(* Logix 5000 project; controller PRU vendor 1 type 14 code 107 rev 20.13; software revision 20.01; part 11 of 17 *)
(* tags used below, declared in another part *)
   AFI : BOOL;
   CHANGING_TOTE : BOOL;
   CHANGING_TOTE_1 : BOOL;
   CHANGING_TOTE_2 : BOOL;
   CHANGING_TOTE_3 : BOOL;
   CHANGING_TOTE_4 : BOOL;
   CHANGING_TOTE_5 : BOOL;
   COOL_VFD_Message : MESSAGE;
   DI0_ION : BOOL;
   DI10_ION : BOOL;
   DI11_ION : BOOL;
   DI12_ION : BOOL;
   DI13_ION : BOOL;
   DI14_ION : BOOL;
   DI15_ION : BOOL;
   DI16_ION : BOOL;
   DI17_ION : BOOL;
   DI18_ION : BOOL;
   DI19_ION : BOOL;
   DI1_ION : BOOL;
   DI20_ION : BOOL;
   DI21_ION : BOOL;
   DI22_ION : BOOL;
   DI23_ION : BOOL;
   DI24_ION : BOOL;
   DI25_ION : BOOL;
   DI26_ION : BOOL;
   DI27_ION : BOOL;
   DI28_ION : BOOL;
   DI29_ION : BOOL;
   DI2_ION : BOOL;
   DI30_ION : BOOL;
   DI31_ION : BOOL;
   DI3_ION : BOOL;
   DI4_ION : BOOL;
   DI5_ION : BOOL;
   DI6_ION : BOOL;
   DI7_ION : BOOL;
   DI8_ION : BOOL;
   DI9_ION : BOOL;
   DUMMY_REAL : REAL;
   ESR_CONTACT_1_ION : BOOL;
   ESR_CONTACT_2_ION : BOOL;
   ESR_CONTACT_3_ION : BOOL;
   ESR_RESET_PB_ION : BOOL;
   ESTOP_PB_IOF : BOOL;   // E-STOP PUSHBUTTON IS PUSHED.
   FAULT : DINT[100];
   FS0101_ION : BOOL;   // LOW FLOW SWITCH - INLET AND DISCHARGE PURGE
   FS0102H_ION : BOOL;   // HIGH FLOW SWITCH - DISCHARGE END SHAFT SEAL
   FS0102L_ION : BOOL;   // LOW FLOW SWITCH - DISCHARGE END SHAFT SEAL
   FS0103H_ION : BOOL;   // HIGH FLOW SWITCH - CHAMBER END INLET SEALS
   FS0103L_ION : BOOL;   // LOW FLOW SWITCH - CHAMBER END INLET SEALS
   FS0201_ION : BOOL;   // LOW FLOW SWITCH - KG021 PURGE
   FS0202_ION : BOOL;   // LOW FLOW SWITCH - KG022 PURGE
   FS0203H_ION : BOOL;   // HIGH FLOW SWITCH - COOLING SHAFT SEALS
   FS0203L_ION : BOOL;   // LOW FLOW SWITCH - COOLING SHAFT SEALS
   FS0204_ION : BOOL;   // LOW FLOW SWITCH - COOLING SCREW COOLING WATER
   HEATER_1_ALARM_ION : BOOL;
   HEATER_2_ALARM_ION : BOOL;
   HEATER_3_ALARM_ION : BOOL;
   HEATER_4_ALARM_ION : BOOL;
   HEATER_5_ALARM_ION : BOOL;
   HMI_ALARM_RESET : BOOL;
   HMI_ALARM_RESET_ONS : BOOL;
   HMI_ALARM_RESET_PB : BOOL;
   HMI_ALARM_RESET_TOF : TIMER;
   HMI_ALARM_RESET_TON : TIMER;
   HMI_COOL_MOTOR : INT;
   HMI_COOL_MOTOR_PRE : INT;
   HMI_DI0_FORCE_OFF : BOOL;
   HMI_DI0_FORCE_ON : BOOL;
   HMI_DI10_FORCE_OFF : BOOL;
   HMI_DI10_FORCE_ON : BOOL;
   HMI_DI11_FORCE_OFF : BOOL;
   HMI_DI11_FORCE_ON : BOOL;
   HMI_DI12_FORCE_OFF : BOOL;
   HMI_DI12_FORCE_ON : BOOL;
   HMI_DI13_FORCE_OFF : BOOL;
   HMI_DI13_FORCE_ON : BOOL;
   HMI_DI14_FORCE_OFF : BOOL;
   HMI_DI14_FORCE_ON : BOOL;
   HMI_DI15_FORCE_OFF : BOOL;
   HMI_DI15_FORCE_ON : BOOL;
   HMI_DI16_FORCE_OFF : BOOL;
   HMI_DI16_FORCE_ON : BOOL;
   HMI_DI17_FORCE_OFF : BOOL;
   HMI_DI17_FORCE_ON : BOOL;
   HMI_DI18_FORCE_OFF : BOOL;
   HMI_DI18_FORCE_ON : BOOL;
   HMI_DI19_FORCE_OFF : BOOL;
   HMI_DI19_FORCE_ON : BOOL;
   HMI_DI1_FORCE_OFF : BOOL;
   HMI_DI1_FORCE_ON : BOOL;
   HMI_DI20_FORCE_OFF : BOOL;
   HMI_DI20_FORCE_ON : BOOL;
   HMI_DI21_FORCE_OFF : BOOL;
   HMI_DI21_FORCE_ON : BOOL;
   HMI_DI22_FORCE_OFF : BOOL;
   HMI_DI22_FORCE_ON : BOOL;
   HMI_DI23_FORCE_OFF : BOOL;
   HMI_DI23_FORCE_ON : BOOL;
   HMI_DI24_FORCE_OFF : BOOL;
   HMI_DI24_FORCE_ON : BOOL;
   HMI_DI25_FORCE_OFF : BOOL;
   HMI_DI25_FORCE_ON : BOOL;
   HMI_DI26_FORCE_OFF : BOOL;
   HMI_DI26_FORCE_ON : BOOL;
   HMI_DI27_FORCE_OFF : BOOL;
   HMI_DI27_FORCE_ON : BOOL;
   HMI_DI28_FORCE_OFF : BOOL;
   HMI_DI28_FORCE_ON : BOOL;
   HMI_DI29_FORCE_OFF : BOOL;
   HMI_DI29_FORCE_ON : BOOL;
   HMI_DI2_FORCE_OFF : BOOL;
   HMI_DI2_FORCE_ON : BOOL;
   HMI_DI30_FORCE_OFF : BOOL;
   HMI_DI30_FORCE_ON : BOOL;
   HMI_DI31_FORCE_OFF : BOOL;
   HMI_DI31_FORCE_ON : BOOL;
   HMI_DI3_FORCE_OFF : BOOL;
   HMI_DI3_FORCE_ON : BOOL;
   HMI_DI4_FORCE_OFF : BOOL;
   HMI_DI4_FORCE_ON : BOOL;
   HMI_DI5_FORCE_OFF : BOOL;
   HMI_DI5_FORCE_ON : BOOL;
   HMI_DI6_FORCE_OFF : BOOL;
   HMI_DI6_FORCE_ON : BOOL;
   HMI_DI7_FORCE_OFF : BOOL;
   HMI_DI7_FORCE_ON : BOOL;
   HMI_DI8_FORCE_OFF : BOOL;
   HMI_DI8_FORCE_ON : BOOL;
   HMI_DI9_FORCE_OFF : BOOL;
   HMI_DI9_FORCE_ON : BOOL;
   HMI_DML_MOTOR : INT;
   HMI_DML_MOTOR_PRE : INT;
   HMI_DMR_MOTOR : INT;
   HMI_DMR_MOTOR_PRE : INT;
   K0621_ALARM_ION : BOOL;
   K0621_IS_CLOSED : BOOL;
   K0621_IS_LOCAL : BOOL;
   K0621_IS_OPEN : BOOL;
   K0621_IS_REMOTE : BOOL;
   K0622_ALARM_ION : BOOL;
   K0622_IS_CLOSED : BOOL;
   K0622_IS_LOCAL : BOOL;
   K0622_IS_OPEN : BOOL;
   K0622_IS_REMOTE : BOOL;
   MSG_ONS3 : BOOL;
   ONE_SEC : BOOL;   // 50% Duty Cycle
   ONE_SEC_ONS : BOOL;
   ONE_SEC_SS : BOOL;
   PLC_Time : DINT[8];
   PS0101_ION : BOOL;   // PRESSURE SWITCH - CONTROL PANEL Y/Z N2 PURGE
   PS0102_ION : BOOL;   // PRESSURE SWITCH - MAIN N2 SUPPLY
   PVTIME_OSC_1 : TIMER;
   PVTIME_OSC_2 : TIMER;
   PVTIME_UPDATE : BOOL;
   RESUME_DISCHARGE : BOOL;
   START_TOTE_CHANGE : BOOL;
   TE0101 : REAL;
   TE0101_SEL_ION : BOOL;
   TE0102 : REAL;
   TE0102_SEL_ION : BOOL;
   TE0103 : REAL;
   TE0103_SEL_ION : BOOL;
   TE0104 : REAL;
   TE0104_SEL_ION : BOOL;
   TE0105 : REAL;
   TE0105_SEL_ION : BOOL;
   TE0106 : REAL;
   TE0106_SEL_ION : BOOL;
   TE0107 : REAL;
   TE0107_SEL_ION : BOOL;
   TE0108 : REAL;
   TE0108_SEL_ION : BOOL;
   TE0109 : REAL;
   TE0109_SEL_ION : BOOL;
   TE0110 : REAL;
   TE0110_SEL_ION : BOOL;
   TE0111 : REAL;
   TE0111_SEL_ION : BOOL;
   TE0112 : REAL;
   TE0112_SEL_ION : BOOL;
   TE0113 : REAL;
   TE0113_SEL_ION : BOOL;
   TE0114 : REAL;
   TE0114_SEL_ION : BOOL;
   TE0115 : REAL;
   TE0115_SEL_ION : BOOL;
   TE0116 : REAL;
   TE0116_SEL_ION : BOOL;
   TE0117 : REAL;
   TE0117_SEL_ION : BOOL;
   TE0118 : REAL;
   TE0118_SEL_ION : BOOL;
   TE0119 : REAL;
   TE0119_SEL_ION : BOOL;
   TE0120 : REAL;
   TE0120_SEL_ION : BOOL;
   TE0121 : REAL;
   TE0121_SEL_ION : BOOL;
   TE0122 : REAL;
   TE0122_SEL_ION : BOOL;
   TE0123 : REAL;
   TE0123_SEL_ION : BOOL;
   TE0124 : REAL;
   TE0124_SEL_ION : BOOL;
   TE0125 : REAL;
   TE0125_SEL_ION : BOOL;
   TE0126 : REAL;
   TE0126_SEL_ION : BOOL;
   TE0127 : REAL;
   TE0127_SEL_ION : BOOL;
   TE0128 : REAL;
   TE0128_SEL_ION : BOOL;
   TE0129 : REAL;
   TE0129_SEL_ION : BOOL;
   TE0130 : REAL;
   TE0130_SEL_ION : BOOL;
   TIMER_MSG_OFF : TIMER;
   TIMER_MSG_ON : TIMER;
   TIMER_ONE_SEC_OFF : TIMER;
   TIMER_ONE_SEC_ON : TIMER;
   TIMER_WDT_OFF : TIMER;
   TIMER_WDT_ON : TIMER;
   TOTE_CHANGE_MODE : INT;
   TOTE_CHANGE_REMAINING : REAL;
   TOTE_CHANGE_TIMED_OUT : BOOL;
   TOTE_CHANGEOUT_TOF : TIMER;
   TOTE_CHANGEOUT_TON : TIMER;
   VFD_3_Current : DINT;
   VFD_3_Current_Real : REAL;
   VFD_3_Tot : EnergyTot;   // Cooling Screw
   VFD_AUTO_RESET : BOOL;
   WDT_ONS : BOOL;
   WDT_SS : BOOL;
   ZONE_1_SELECT_TE : TE_SELECTED_AVE;
   ZONE_1_TEMP_AVE : DINT;
   ZONE_2_SELECT_TE : TE_SELECTED_AVE;
   ZONE_2_TEMP_AVE : REAL;
   ZONE_3_SELECT_TE : TE_SELECTED_AVE;
   ZONE_3_TEMP_AVE : REAL;
   ZONE_4_SELECT_TE : TE_SELECTED_AVE;
   ZONE_4_TEMP_AVE : REAL;
   ZONE_5_SELECT_TE : TE_SELECTED_AVE;
   ZONE_5_TEMP_AVE : REAL;
   ZONE_6_SELECT_TE : TE_SELECTED_AVE;
   ZONE_6_TEMP_AVE : REAL;
   ZONE_7_SELECT_TE : TE_SELECTED_AVE;
   ZONE_7_TEMP_AVE : REAL;
(* MainProgram, continued *)

ROUTINE C04_ZONE_TEMPS   (* ladder *)
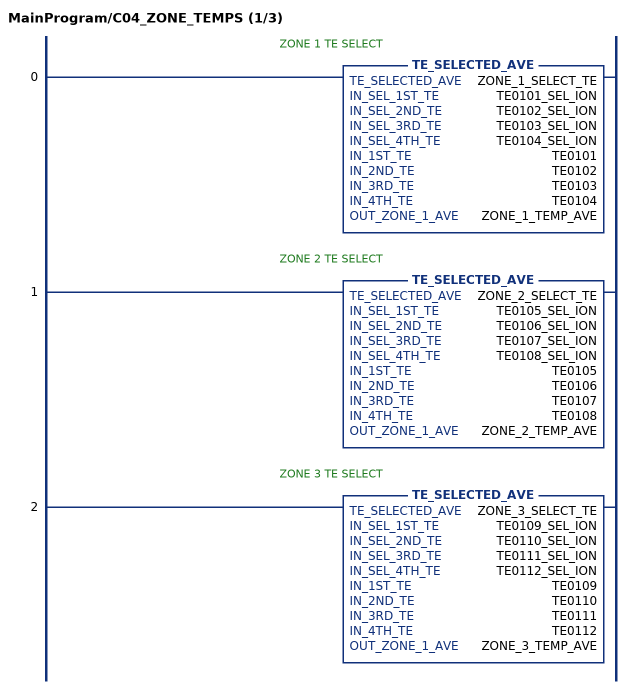
   // ZONE 1 TE SELECT
   0: TE_SELECTED_AVE(ZONE_1_SELECT_TE,TE0101_SEL_ION,TE0102_SEL_ION,TE0103_SEL_ION,TE0104_SEL_ION,TE0101,TE0102,TE0103,TE0104,ZONE_1_TEMP_AVE);
   // ZONE 2 TE SELECT
   1: TE_SELECTED_AVE(ZONE_2_SELECT_TE,TE0105_SEL_ION,TE0106_SEL_ION,TE0107_SEL_ION,TE0108_SEL_ION,TE0105,TE0106,TE0107,TE0108,ZONE_2_TEMP_AVE);
   // ZONE 3 TE SELECT
   2: TE_SELECTED_AVE(ZONE_3_SELECT_TE,TE0109_SEL_ION,TE0110_SEL_ION,TE0111_SEL_ION,TE0112_SEL_ION,TE0109,TE0110,TE0111,TE0112,ZONE_3_TEMP_AVE);
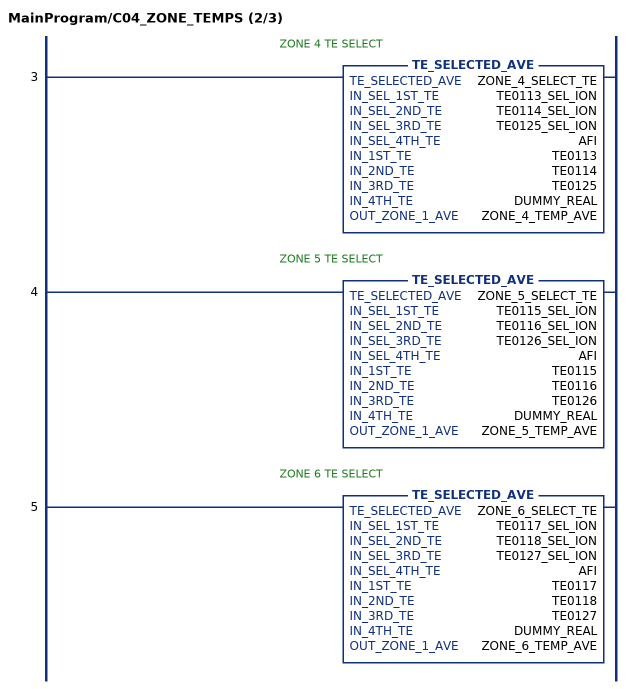
   // ZONE 4 TE SELECT
   3: TE_SELECTED_AVE(ZONE_4_SELECT_TE,TE0113_SEL_ION,TE0114_SEL_ION,TE0125_SEL_ION,AFI,TE0113,TE0114,TE0125,DUMMY_REAL,ZONE_4_TEMP_AVE);
   // ZONE 5 TE SELECT
   4: TE_SELECTED_AVE(ZONE_5_SELECT_TE,TE0115_SEL_ION,TE0116_SEL_ION,TE0126_SEL_ION,AFI,TE0115,TE0116,TE0126,DUMMY_REAL,ZONE_5_TEMP_AVE);
   // ZONE 6 TE SELECT
   5: TE_SELECTED_AVE(ZONE_6_SELECT_TE,TE0117_SEL_ION,TE0118_SEL_ION,TE0127_SEL_ION,AFI,TE0117,TE0118,TE0127,DUMMY_REAL,ZONE_6_TEMP_AVE);
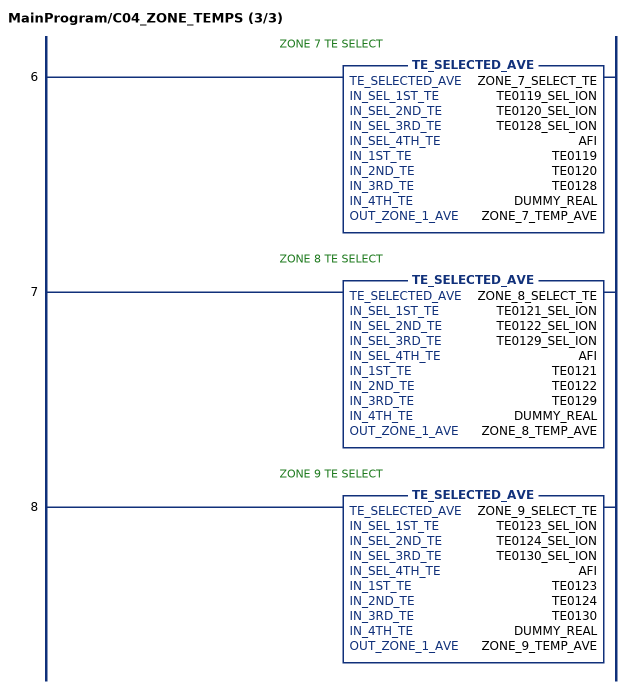
   // ZONE 7 TE SELECT
   6: TE_SELECTED_AVE(ZONE_7_SELECT_TE,TE0119_SEL_ION,TE0120_SEL_ION,TE0128_SEL_ION,AFI,TE0119,TE0120,TE0128,DUMMY_REAL,ZONE_7_TEMP_AVE);
   // ZONE 8 TE SELECT
   7: TE_SELECTED_AVE(ZONE_8_SELECT_TE,TE0121_SEL_ION,TE0122_SEL_ION,TE0129_SEL_ION,AFI,TE0121,TE0122,TE0129,DUMMY_REAL,ZONE_8_TEMP_AVE);
   // ZONE 9 TE SELECT
   8: TE_SELECTED_AVE(ZONE_9_SELECT_TE,TE0123_SEL_ION,TE0124_SEL_ION,TE0130_SEL_ION,AFI,TE0123,TE0124,TE0130,DUMMY_REAL,ZONE_9_TEMP_AVE);
END_ROUTINE

ROUTINE C05_TOTE_CHANGE   (* ladder *)
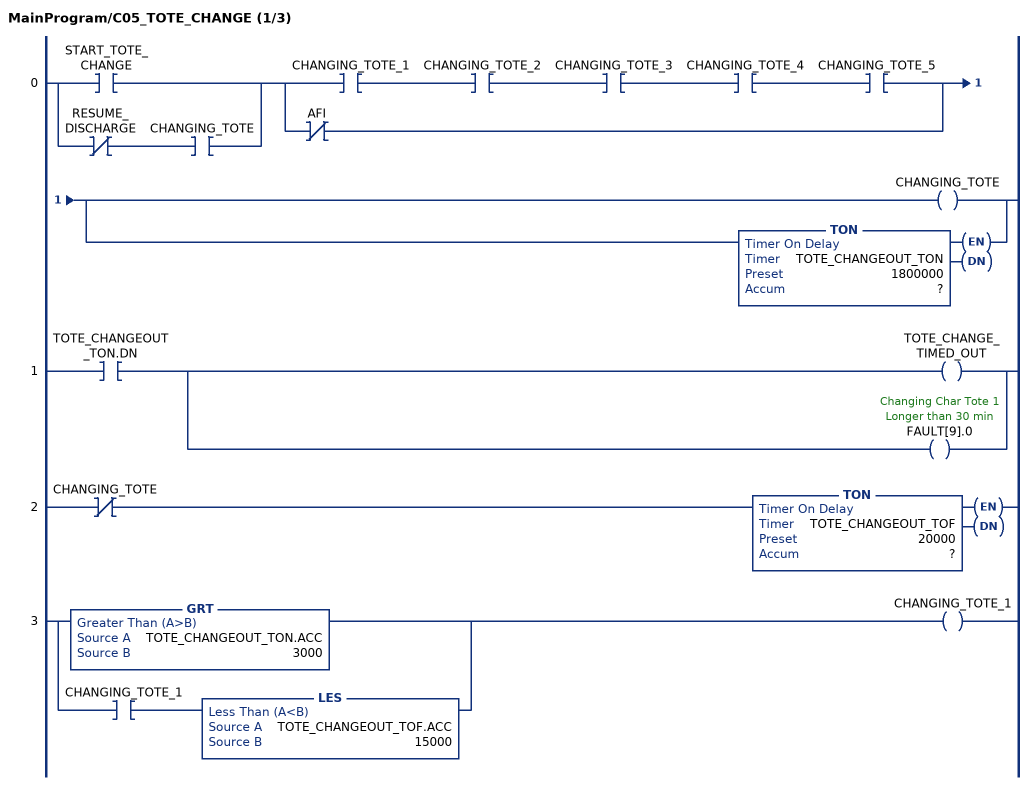
   0: [XIC(START_TOTE_CHANGE) ,XIO(RESUME_DISCHARGE) XIC(CHANGING_TOTE) ][XIC(CHANGING_TOTE_1) XIC(CHANGING_TOTE_2) XIC(CHANGING_TOTE_3) XIC(CHANGING_TOTE_4) XIC(CHANGING_TOTE_5) ,XIO(AFI) ][OTE(CHANGING_TOTE) ,TON(TOTE_CHANGEOUT_TON,?,?) ];
   1: XIC(TOTE_CHANGEOUT_TON.DN)[OTE(TOTE_CHANGE_TIMED_OUT) ,OTE(FAULT[9].0) ];
   2: XIO(CHANGING_TOTE)TON(TOTE_CHANGEOUT_TOF,?,?);
   3: [GRT(TOTE_CHANGEOUT_TON.ACC,3000) ,XIC(CHANGING_TOTE_1) LES(TOTE_CHANGEOUT_TOF.ACC,15000) ]OTE(CHANGING_TOTE_1);
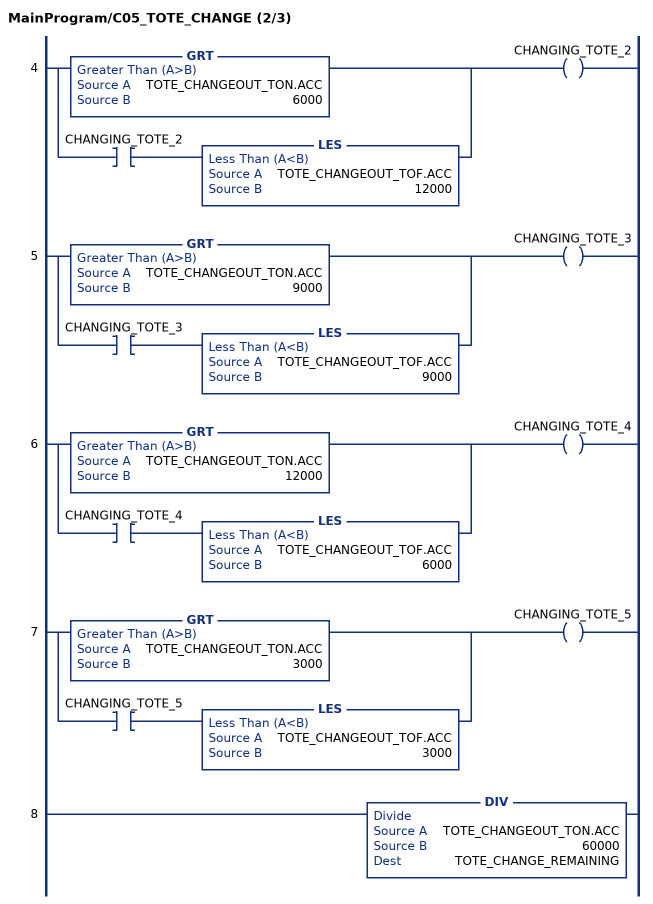
   4: [GRT(TOTE_CHANGEOUT_TON.ACC,6000) ,XIC(CHANGING_TOTE_2) LES(TOTE_CHANGEOUT_TOF.ACC,12000) ]OTE(CHANGING_TOTE_2);
   5: [GRT(TOTE_CHANGEOUT_TON.ACC,9000) ,XIC(CHANGING_TOTE_3) LES(TOTE_CHANGEOUT_TOF.ACC,9000) ]OTE(CHANGING_TOTE_3);
   6: [GRT(TOTE_CHANGEOUT_TON.ACC,12000) ,XIC(CHANGING_TOTE_4) LES(TOTE_CHANGEOUT_TOF.ACC,6000) ]OTE(CHANGING_TOTE_4);
   7: [GRT(TOTE_CHANGEOUT_TON.ACC,3000) ,XIC(CHANGING_TOTE_5) LES(TOTE_CHANGEOUT_TOF.ACC,3000) ]OTE(CHANGING_TOTE_5);
   8: DIV(TOTE_CHANGEOUT_TON.ACC,60000,TOTE_CHANGE_REMAINING);
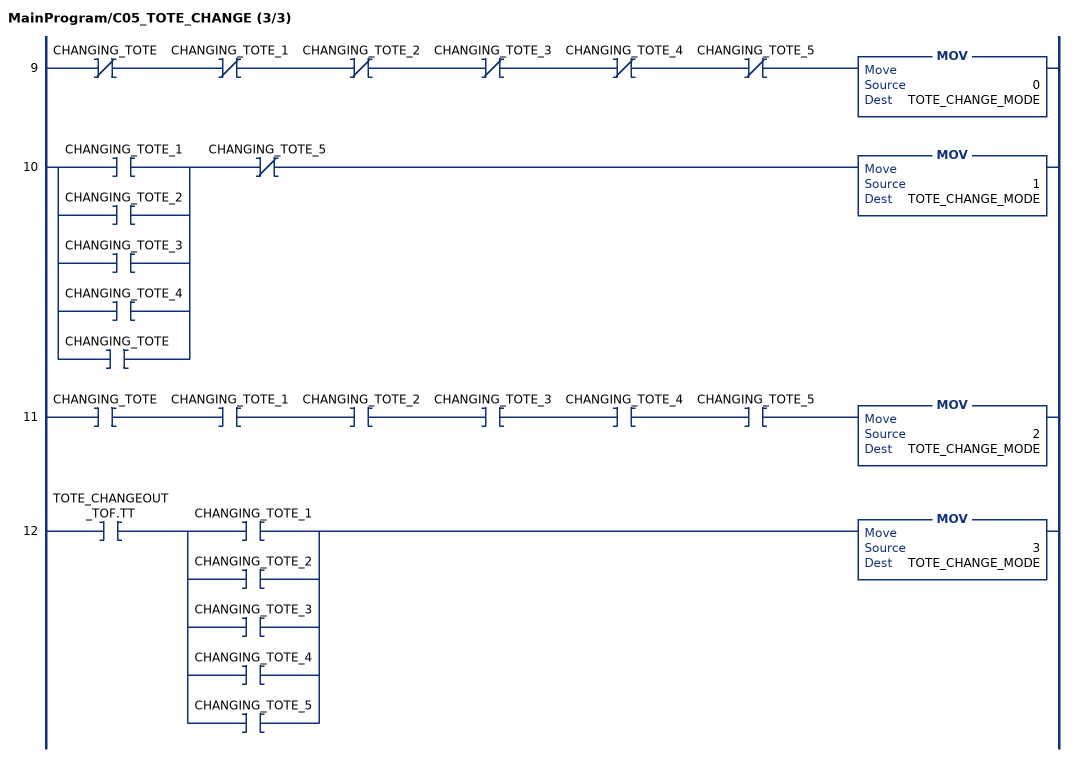
   9: XIO(CHANGING_TOTE)XIO(CHANGING_TOTE_1)XIO(CHANGING_TOTE_2)XIO(CHANGING_TOTE_3)XIO(CHANGING_TOTE_4)XIO(CHANGING_TOTE_5)MOV(0,TOTE_CHANGE_MODE);
   10: [XIC(CHANGING_TOTE_1) ,XIC(CHANGING_TOTE_2) ,XIC(CHANGING_TOTE_3) ,XIC(CHANGING_TOTE_4) ,XIC(CHANGING_TOTE) ]XIO(CHANGING_TOTE_5)MOV(1,TOTE_CHANGE_MODE);
   11: XIC(CHANGING_TOTE)XIC(CHANGING_TOTE_1)XIC(CHANGING_TOTE_2)XIC(CHANGING_TOTE_3)XIC(CHANGING_TOTE_4)XIC(CHANGING_TOTE_5)MOV(2,TOTE_CHANGE_MODE);
   12: XIC(TOTE_CHANGEOUT_TOF.TT)[XIC(CHANGING_TOTE_1) ,XIC(CHANGING_TOTE_2) ,XIC(CHANGING_TOTE_3) ,XIC(CHANGING_TOTE_4) ,XIC(CHANGING_TOTE_5) ]MOV(3,TOTE_CHANGE_MODE);
END_ROUTINE

ROUTINE E00_Overhead   (* ladder *)
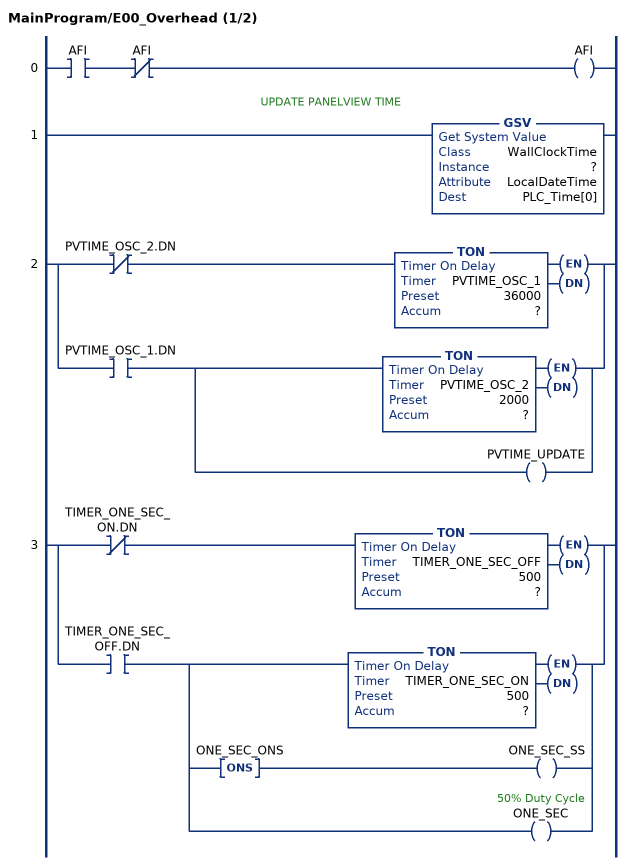
   0: XIC(AFI)XIO(AFI)OTE(AFI);
   // UPDATE PANELVIEW TIME
   1: GSV(WallClockTime,?,LocalDateTime,PLC_Time[0]);
   2: [XIO(PVTIME_OSC_2.DN) TON(PVTIME_OSC_1,?,?) ,XIC(PVTIME_OSC_1.DN) [TON(PVTIME_OSC_2,?,?) ,OTE(PVTIME_UPDATE) ] ];
   3: [XIO(TIMER_ONE_SEC_ON.DN) TON(TIMER_ONE_SEC_OFF,?,?) ,XIC(TIMER_ONE_SEC_OFF.DN) [TON(TIMER_ONE_SEC_ON,?,?) ,ONS(ONE_SEC_ONS) OTE(ONE_SEC_SS) ,OTE(ONE_SEC) ] ];
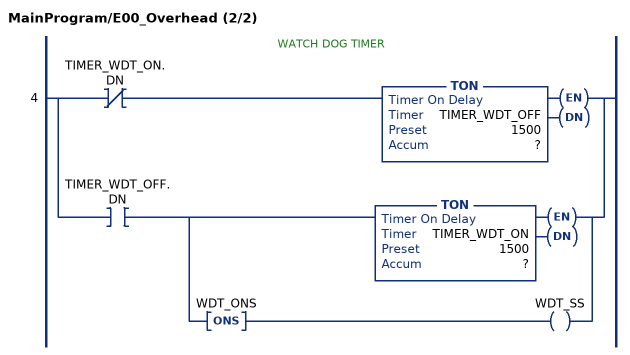
   // WATCH DOG TIMER
   4: [XIO(TIMER_WDT_ON.DN) TON(TIMER_WDT_OFF,?,?) ,XIC(TIMER_WDT_OFF.DN) [TON(TIMER_WDT_ON,?,?) ,ONS(WDT_ONS) OTE(WDT_SS) ] ];
END_ROUTINE

ROUTINE F00_HMI   (* ladder *)
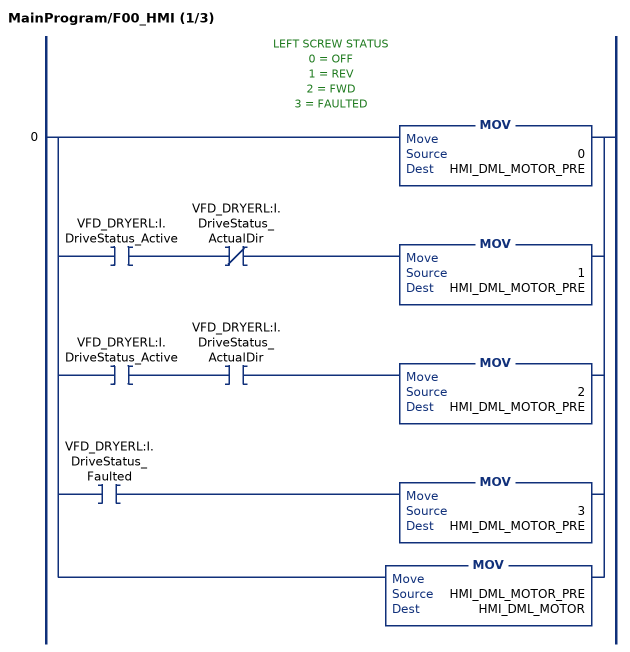
   // LEFT SCREW STATUS
   // 0 = OFF
   // 1 = REV
   // 2 = FWD
   // 3 = FAULTED
   0: [MOV(0,HMI_DML_MOTOR_PRE) ,XIC(VFD_DRYERL:I.DriveStatus_Active) XIO(VFD_DRYERL:I.DriveStatus_ActualDir) MOV(1,HMI_DML_MOTOR_PRE) ,XIC(VFD_DRYERL:I.DriveStatus_Active) XIC(VFD_DRYERL:I.DriveStatus_ActualDir) MOV(2,HMI_DML_MOTOR_PRE) ,XIC(VFD_DRYERL:I.DriveStatus_Faulted) MOV(3,HMI_DML_MOTOR_PRE) ,MOV(HMI_DML_MOTOR_PRE,HMI_DML_MOTOR) ];
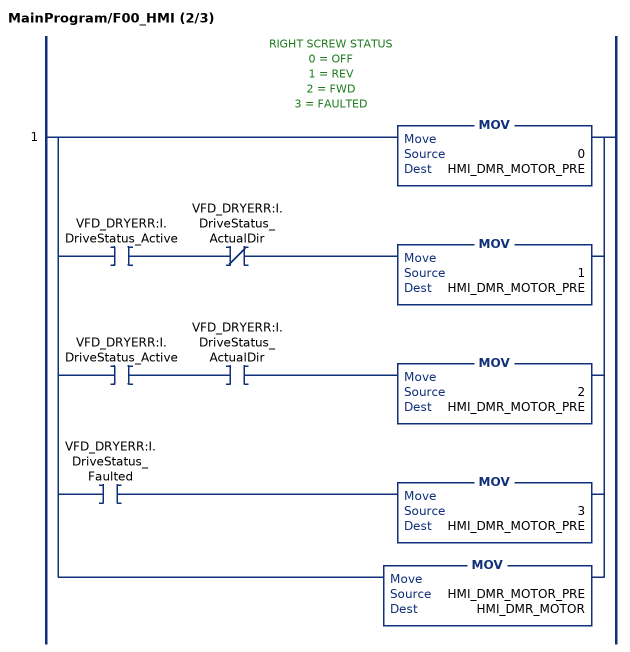
   // RIGHT SCREW STATUS
   // 0 = OFF
   // 1 = REV
   // 2 = FWD
   // 3 = FAULTED
   1: [MOV(0,HMI_DMR_MOTOR_PRE) ,XIC(VFD_DRYERR:I.DriveStatus_Active) XIO(VFD_DRYERR:I.DriveStatus_ActualDir) MOV(1,HMI_DMR_MOTOR_PRE) ,XIC(VFD_DRYERR:I.DriveStatus_Active) XIC(VFD_DRYERR:I.DriveStatus_ActualDir) MOV(2,HMI_DMR_MOTOR_PRE) ,XIC(VFD_DRYERR:I.DriveStatus_Faulted) MOV(3,HMI_DMR_MOTOR_PRE) ,MOV(HMI_DMR_MOTOR_PRE,HMI_DMR_MOTOR) ];
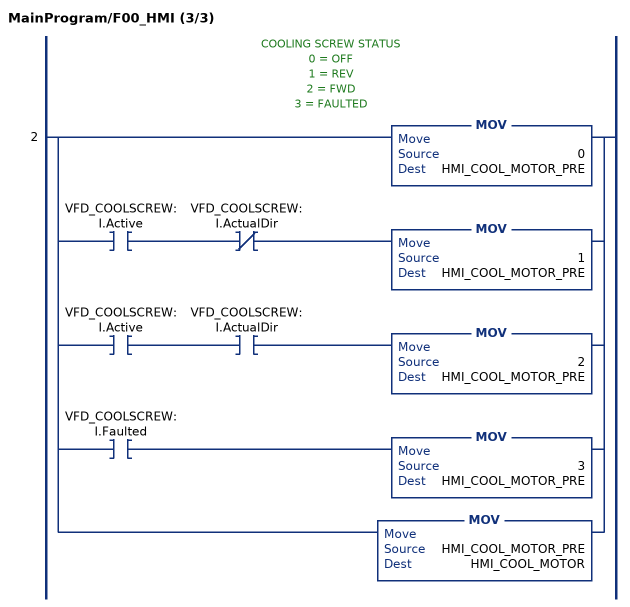
   // COOLING SCREW STATUS
   // 0 = OFF
   // 1 = REV
   // 2 = FWD
   // 3 = FAULTED
   2: [MOV(0,HMI_COOL_MOTOR_PRE) ,XIC(VFD_COOLSCREW:I.Active) XIO(VFD_COOLSCREW:I.ActualDir) MOV(1,HMI_COOL_MOTOR_PRE) ,XIC(VFD_COOLSCREW:I.Active) XIC(VFD_COOLSCREW:I.ActualDir) MOV(2,HMI_COOL_MOTOR_PRE) ,XIC(VFD_COOLSCREW:I.Faulted) MOV(3,HMI_COOL_MOTOR_PRE) ,MOV(HMI_COOL_MOTOR_PRE,HMI_COOL_MOTOR) ];
END_ROUTINE

ROUTINE F01_VFD_Msgs_Reset   (* ladder *)
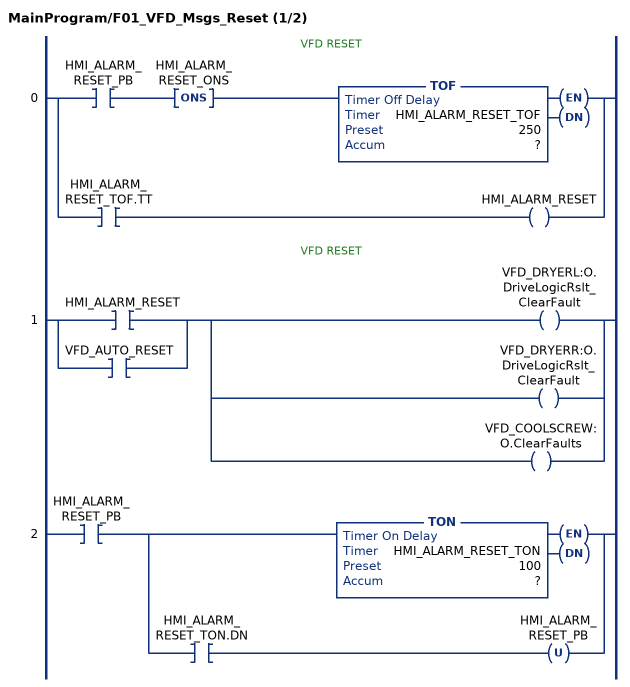
   // VFD RESET
   0: [XIC(HMI_ALARM_RESET_PB) ONS(HMI_ALARM_RESET_ONS) TOF(HMI_ALARM_RESET_TOF,?,?) ,XIC(HMI_ALARM_RESET_TOF.TT) OTE(HMI_ALARM_RESET) ];
   // VFD RESET
   1: [XIC(HMI_ALARM_RESET) ,XIC(VFD_AUTO_RESET) ][OTE(VFD_DRYERL:O.DriveLogicRslt_ClearFault) ,OTE(VFD_DRYERR:O.DriveLogicRslt_ClearFault) ,OTE(VFD_COOLSCREW:O.ClearFaults) ];
   2: XIC(HMI_ALARM_RESET_PB)[TON(HMI_ALARM_RESET_TON,?,?) ,XIC(HMI_ALARM_RESET_TON.DN) OTU(HMI_ALARM_RESET_PB) ];
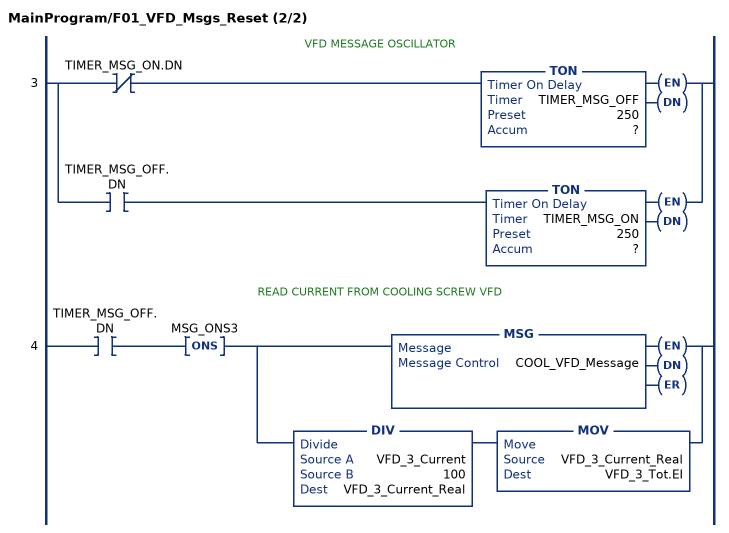
   // VFD MESSAGE OSCILLATOR
   3: [XIO(TIMER_MSG_ON.DN) TON(TIMER_MSG_OFF,?,?) ,XIC(TIMER_MSG_OFF.DN) TON(TIMER_MSG_ON,?,?) ];
   // READ CURRENT FROM COOLING SCREW VFD
   4: XIC(TIMER_MSG_OFF.DN)ONS(MSG_ONS3)[MSG(COOL_VFD_Message) ,DIV(VFD_3_Current,100,VFD_3_Current_Real) MOV(VFD_3_Current_Real,VFD_3_Tot.EI) ];
END_ROUTINE

ROUTINE G01_MAP_DIG_INPUTS   (* ladder *)
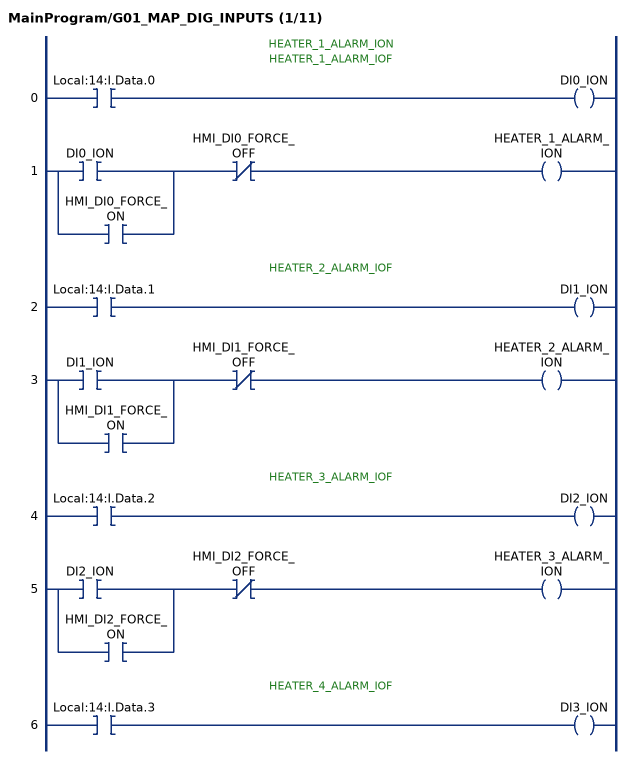
   // HEATER_1_ALARM_ION
   // HEATER_1_ALARM_IOF
   0: XIC(Local:14:I.Data.0)OTE(DI0_ION);
   1: [XIC(DI0_ION) ,XIC(HMI_DI0_FORCE_ON) ]XIO(HMI_DI0_FORCE_OFF)OTE(HEATER_1_ALARM_ION);
   // HEATER_2_ALARM_IOF
   2: XIC(Local:14:I.Data.1)OTE(DI1_ION);
   3: [XIC(DI1_ION) ,XIC(HMI_DI1_FORCE_ON) ]XIO(HMI_DI1_FORCE_OFF)OTE(HEATER_2_ALARM_ION);
   // HEATER_3_ALARM_IOF
   4: XIC(Local:14:I.Data.2)OTE(DI2_ION);
   5: [XIC(DI2_ION) ,XIC(HMI_DI2_FORCE_ON) ]XIO(HMI_DI2_FORCE_OFF)OTE(HEATER_3_ALARM_ION);
   // HEATER_4_ALARM_IOF
   6: XIC(Local:14:I.Data.3)OTE(DI3_ION);
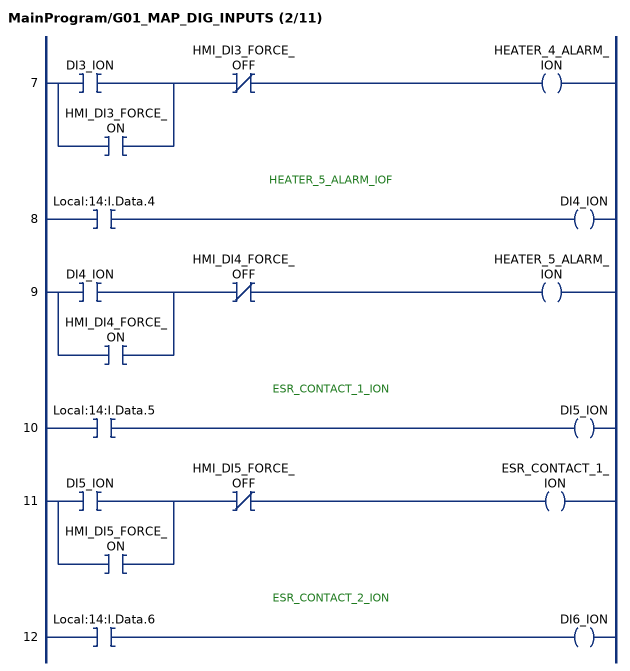
   7: [XIC(DI3_ION) ,XIC(HMI_DI3_FORCE_ON) ]XIO(HMI_DI3_FORCE_OFF)OTE(HEATER_4_ALARM_ION);
   // HEATER_5_ALARM_IOF
   8: XIC(Local:14:I.Data.4)OTE(DI4_ION);
   9: [XIC(DI4_ION) ,XIC(HMI_DI4_FORCE_ON) ]XIO(HMI_DI4_FORCE_OFF)OTE(HEATER_5_ALARM_ION);
   // ESR_CONTACT_1_ION
   10: XIC(Local:14:I.Data.5)OTE(DI5_ION);
   11: [XIC(DI5_ION) ,XIC(HMI_DI5_FORCE_ON) ]XIO(HMI_DI5_FORCE_OFF)OTE(ESR_CONTACT_1_ION);
   // ESR_CONTACT_2_ION
   12: XIC(Local:14:I.Data.6)OTE(DI6_ION);
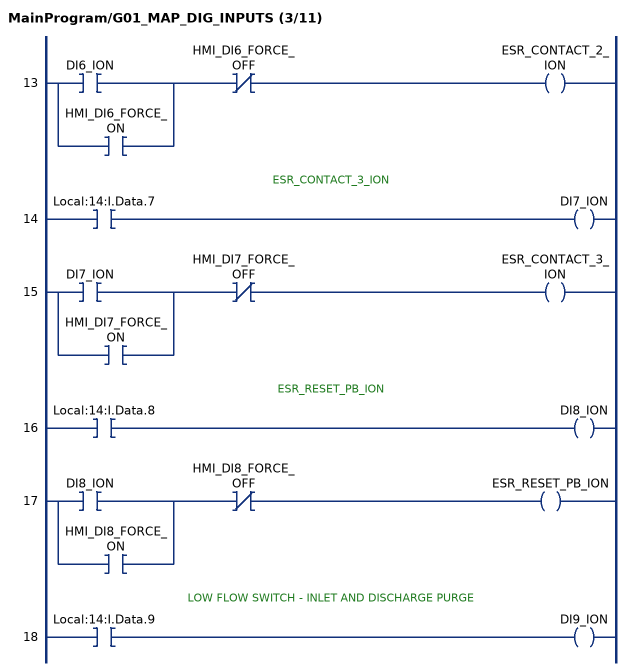
   13: [XIC(DI6_ION) ,XIC(HMI_DI6_FORCE_ON) ]XIO(HMI_DI6_FORCE_OFF)OTE(ESR_CONTACT_2_ION);
   // ESR_CONTACT_3_ION
   14: XIC(Local:14:I.Data.7)OTE(DI7_ION);
   15: [XIC(DI7_ION) ,XIC(HMI_DI7_FORCE_ON) ]XIO(HMI_DI7_FORCE_OFF)OTE(ESR_CONTACT_3_ION);
   // ESR_RESET_PB_ION
   16: XIC(Local:14:I.Data.8)OTE(DI8_ION);
   17: [XIC(DI8_ION) ,XIC(HMI_DI8_FORCE_ON) ]XIO(HMI_DI8_FORCE_OFF)OTE(ESR_RESET_PB_ION);
   // LOW FLOW SWITCH - INLET AND DISCHARGE PURGE
   18: XIC(Local:14:I.Data.9)OTE(DI9_ION);
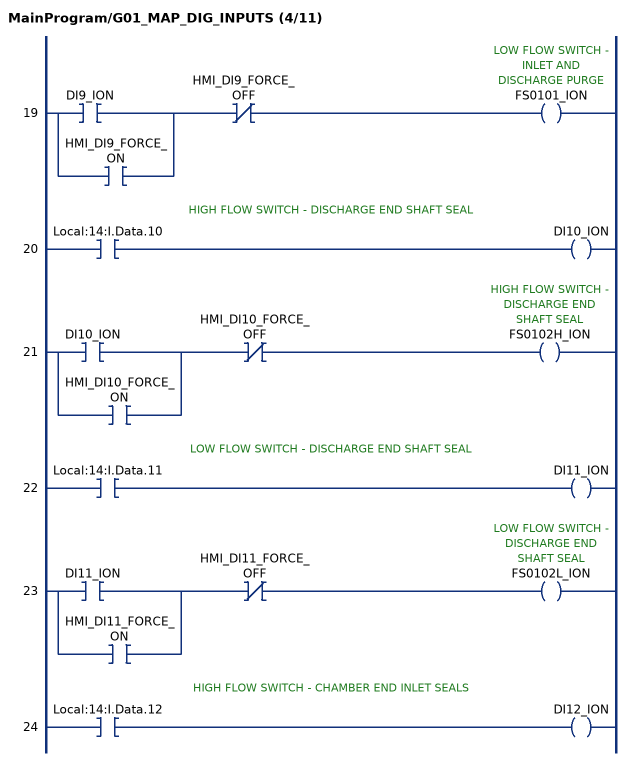
   19: [XIC(DI9_ION) ,XIC(HMI_DI9_FORCE_ON) ]XIO(HMI_DI9_FORCE_OFF)OTE(FS0101_ION);
   // HIGH FLOW SWITCH - DISCHARGE END SHAFT SEAL
   20: XIC(Local:14:I.Data.10)OTE(DI10_ION);
   21: [XIC(DI10_ION) ,XIC(HMI_DI10_FORCE_ON) ]XIO(HMI_DI10_FORCE_OFF)OTE(FS0102H_ION);
   // LOW FLOW SWITCH - DISCHARGE END SHAFT SEAL
   22: XIC(Local:14:I.Data.11)OTE(DI11_ION);
   23: [XIC(DI11_ION) ,XIC(HMI_DI11_FORCE_ON) ]XIO(HMI_DI11_FORCE_OFF)OTE(FS0102L_ION);
   // HIGH FLOW SWITCH - CHAMBER END INLET SEALS
   24: XIC(Local:14:I.Data.12)OTE(DI12_ION);
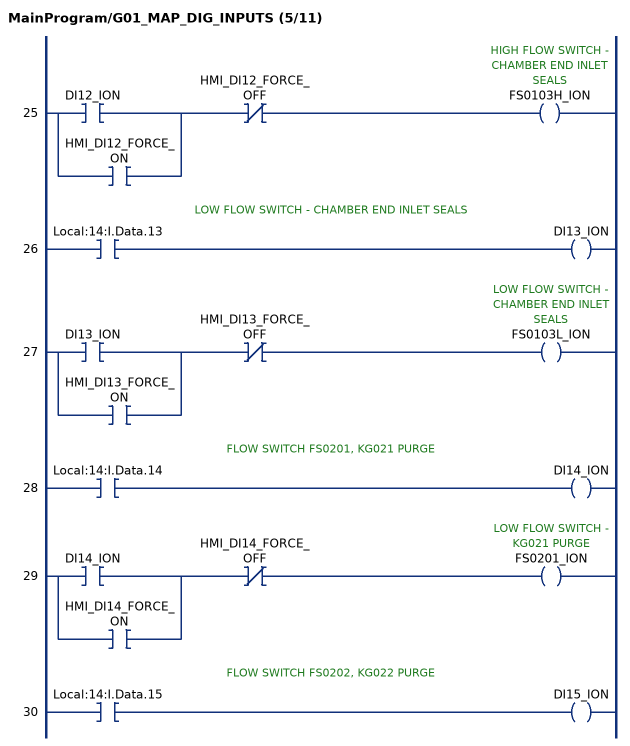
   25: [XIC(DI12_ION) ,XIC(HMI_DI12_FORCE_ON) ]XIO(HMI_DI12_FORCE_OFF)OTE(FS0103H_ION);
   // LOW FLOW SWITCH - CHAMBER END INLET SEALS
   26: XIC(Local:14:I.Data.13)OTE(DI13_ION);
   27: [XIC(DI13_ION) ,XIC(HMI_DI13_FORCE_ON) ]XIO(HMI_DI13_FORCE_OFF)OTE(FS0103L_ION);
   // FLOW SWITCH FS0201, KG021 PURGE
   28: XIC(Local:14:I.Data.14)OTE(DI14_ION);
   29: [XIC(DI14_ION) ,XIC(HMI_DI14_FORCE_ON) ]XIO(HMI_DI14_FORCE_OFF)OTE(FS0201_ION);
   // FLOW SWITCH FS0202, KG022 PURGE
   30: XIC(Local:14:I.Data.15)OTE(DI15_ION);
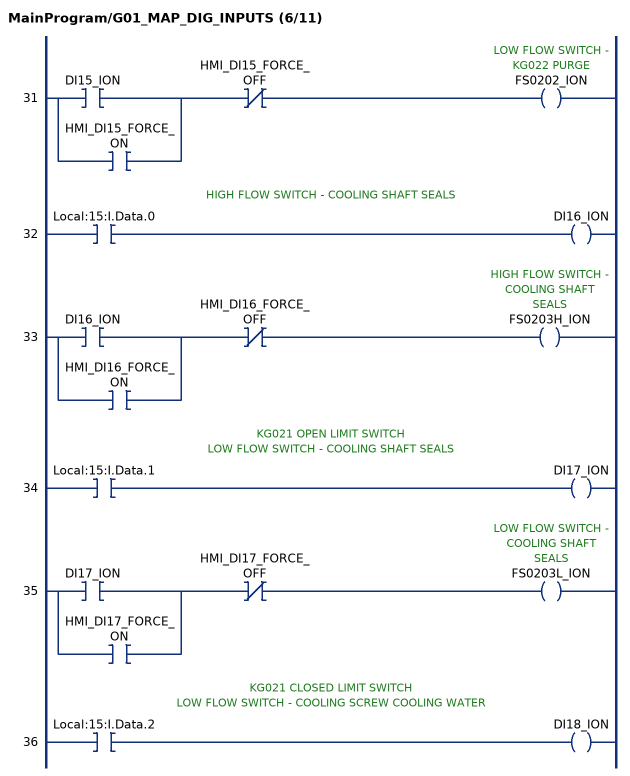
   31: [XIC(DI15_ION) ,XIC(HMI_DI15_FORCE_ON) ]XIO(HMI_DI15_FORCE_OFF)OTE(FS0202_ION);
   // HIGH FLOW SWITCH - COOLING SHAFT SEALS
   32: XIC(Local:15:I.Data.0)OTE(DI16_ION);
   33: [XIC(DI16_ION) ,XIC(HMI_DI16_FORCE_ON) ]XIO(HMI_DI16_FORCE_OFF)OTE(FS0203H_ION);
   // KG021 OPEN LIMIT SWITCH
   // LOW FLOW SWITCH - COOLING SHAFT SEALS
   34: XIC(Local:15:I.Data.1)OTE(DI17_ION);
   35: [XIC(DI17_ION) ,XIC(HMI_DI17_FORCE_ON) ]XIO(HMI_DI17_FORCE_OFF)OTE(FS0203L_ION);
   // KG021 CLOSED LIMIT SWITCH
   // LOW FLOW SWITCH - COOLING SCREW COOLING WATER
   36: XIC(Local:15:I.Data.2)OTE(DI18_ION);
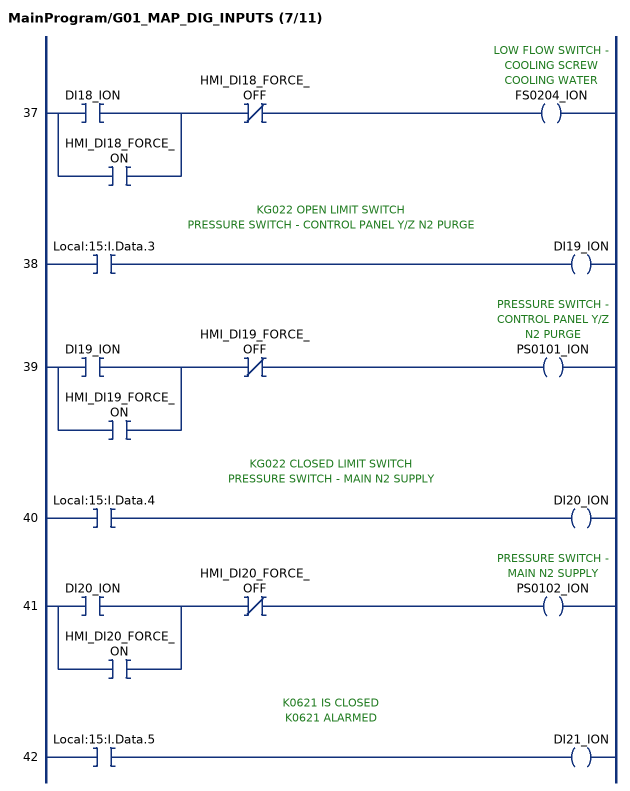
   37: [XIC(DI18_ION) ,XIC(HMI_DI18_FORCE_ON) ]XIO(HMI_DI18_FORCE_OFF)OTE(FS0204_ION);
   // KG022 OPEN LIMIT SWITCH
   // PRESSURE SWITCH - CONTROL PANEL Y/Z N2 PURGE
   38: XIC(Local:15:I.Data.3)OTE(DI19_ION);
   39: [XIC(DI19_ION) ,XIC(HMI_DI19_FORCE_ON) ]XIO(HMI_DI19_FORCE_OFF)OTE(PS0101_ION);
   // KG022 CLOSED LIMIT SWITCH
   // PRESSURE SWITCH - MAIN N2 SUPPLY
   40: XIC(Local:15:I.Data.4)OTE(DI20_ION);
   41: [XIC(DI20_ION) ,XIC(HMI_DI20_FORCE_ON) ]XIO(HMI_DI20_FORCE_OFF)OTE(PS0102_ION);
   // K0621 IS CLOSED
   // K0621 ALARMED
   42: XIC(Local:15:I.Data.5)OTE(DI21_ION);
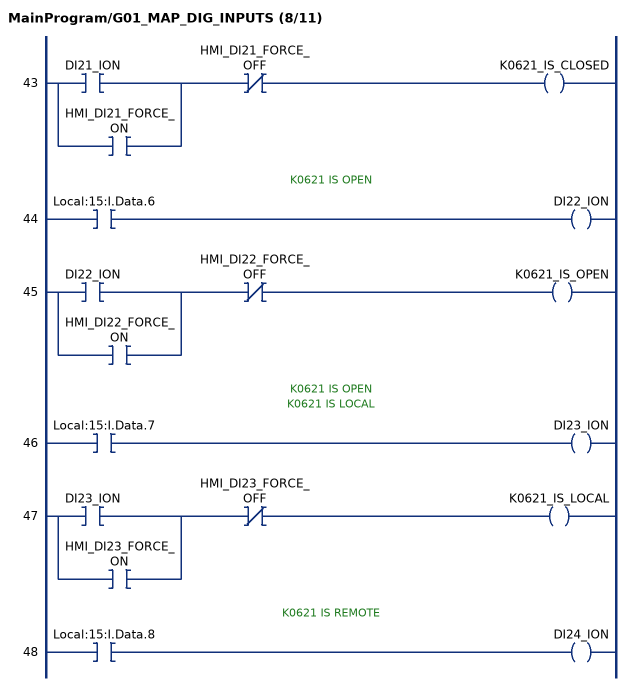
   43: [XIC(DI21_ION) ,XIC(HMI_DI21_FORCE_ON) ]XIO(HMI_DI21_FORCE_OFF)OTE(K0621_IS_CLOSED);
   // K0621 IS OPEN
   44: XIC(Local:15:I.Data.6)OTE(DI22_ION);
   45: [XIC(DI22_ION) ,XIC(HMI_DI22_FORCE_ON) ]XIO(HMI_DI22_FORCE_OFF)OTE(K0621_IS_OPEN);
   // K0621 IS OPEN
   // K0621 IS LOCAL
   46: XIC(Local:15:I.Data.7)OTE(DI23_ION);
   47: [XIC(DI23_ION) ,XIC(HMI_DI23_FORCE_ON) ]XIO(HMI_DI23_FORCE_OFF)OTE(K0621_IS_LOCAL);
   // K0621 IS REMOTE
   48: XIC(Local:15:I.Data.8)OTE(DI24_ION);
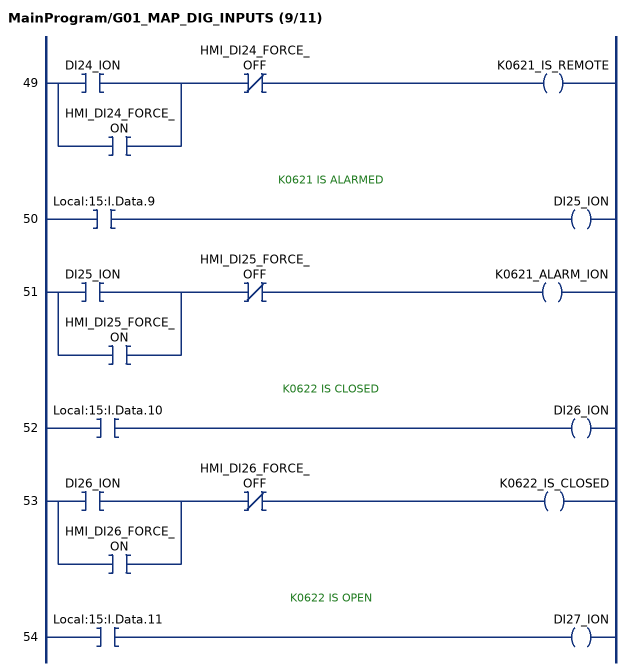
   49: [XIC(DI24_ION) ,XIC(HMI_DI24_FORCE_ON) ]XIO(HMI_DI24_FORCE_OFF)OTE(K0621_IS_REMOTE);
   // K0621 IS ALARMED
   50: XIC(Local:15:I.Data.9)OTE(DI25_ION);
   51: [XIC(DI25_ION) ,XIC(HMI_DI25_FORCE_ON) ]XIO(HMI_DI25_FORCE_OFF)OTE(K0621_ALARM_ION);
   // K0622 IS CLOSED
   52: XIC(Local:15:I.Data.10)OTE(DI26_ION);
   53: [XIC(DI26_ION) ,XIC(HMI_DI26_FORCE_ON) ]XIO(HMI_DI26_FORCE_OFF)OTE(K0622_IS_CLOSED);
   // K0622 IS OPEN
   54: XIC(Local:15:I.Data.11)OTE(DI27_ION);
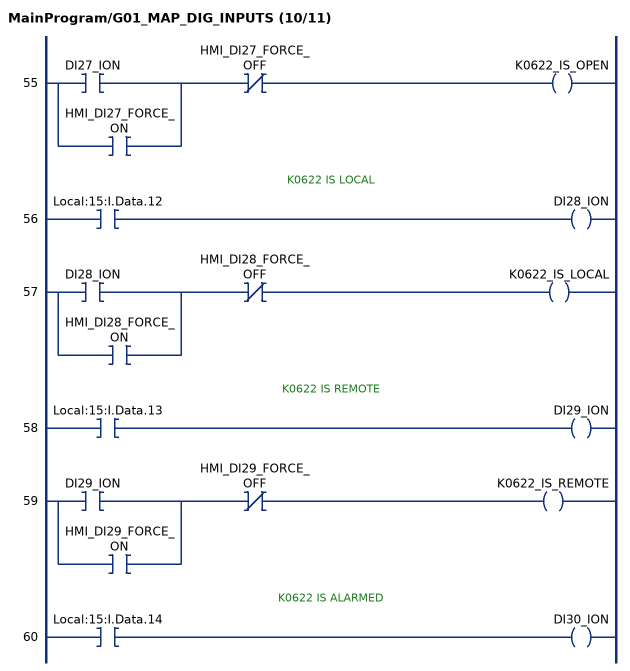
   55: [XIC(DI27_ION) ,XIC(HMI_DI27_FORCE_ON) ]XIO(HMI_DI27_FORCE_OFF)OTE(K0622_IS_OPEN);
   // K0622 IS LOCAL
   56: XIC(Local:15:I.Data.12)OTE(DI28_ION);
   57: [XIC(DI28_ION) ,XIC(HMI_DI28_FORCE_ON) ]XIO(HMI_DI28_FORCE_OFF)OTE(K0622_IS_LOCAL);
   // K0622 IS REMOTE
   58: XIC(Local:15:I.Data.13)OTE(DI29_ION);
   59: [XIC(DI29_ION) ,XIC(HMI_DI29_FORCE_ON) ]XIO(HMI_DI29_FORCE_OFF)OTE(K0622_IS_REMOTE);
   // K0622 IS ALARMED
   60: XIC(Local:15:I.Data.14)OTE(DI30_ION);
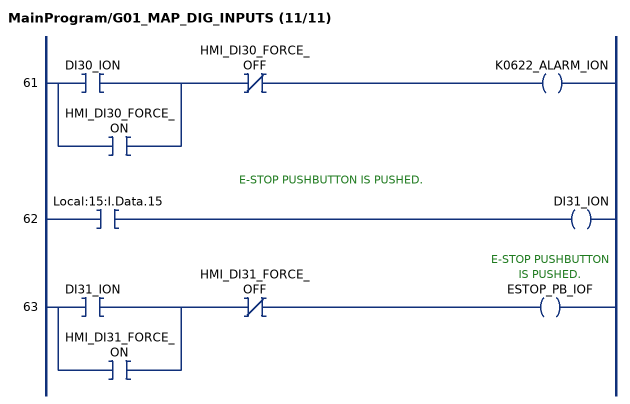
   61: [XIC(DI30_ION) ,XIC(HMI_DI30_FORCE_ON) ]XIO(HMI_DI30_FORCE_OFF)OTE(K0622_ALARM_ION);
   // E-STOP PUSHBUTTON IS PUSHED.
   62: XIC(Local:15:I.Data.15)OTE(DI31_ION);
   63: [XIC(DI31_ION) ,XIC(HMI_DI31_FORCE_ON) ]XIO(HMI_DI31_FORCE_OFF)OTE(ESTOP_PB_IOF);
END_ROUTINE
